TYPE DOXControlCompactChannel :
STRUCT
	{attribute addProperty Name "Control"}
	Control AT %Q* : stDOXcontrolCompact;
END_STRUCT
END_TYPE

(* stored: Version 1.1.0.1, ProductVersion 3.1.4024.9
   DUT DOXControlCompactChannel: Id {8ebbd861-b644-0811-25ec-7e663f4dc605} *)
